    movel([0.494743, -1.360953, -2.580567, -0.770869, 1.570796, 2.065539],accel_mss,speed_ms,0,blend_radius_m)
    movel([0.490867, -1.356572, -2.583531, -0.772287, 1.570796, 2.061664],accel_mss,speed_ms,0,blend_radius_m)
    movel([0.488474, -1.353182, -2.585805, -0.773402, 1.570796, 2.059270],accel_mss,speed_ms,0,blend_radius_m)
    movel([0.485996, -1.348940, -2.588629, -0.774820, 1.570796, 2.056792],accel_mss,speed_ms,0,blend_radius_m)
    movel([0.483593, -1.343799, -2.592018, -0.776572, 1.570796, 2.054390],accel_mss,speed_ms,0,blend_radius_m)
    movel([0.481444, -1.337704, -2.595989, -0.778696, 1.570796, 2.052240],accel_mss,speed_ms,0,blend_radius_m)
    movel([0.480362, -1.333157, -2.598918, -0.780314, 1.570796, 2.051158],accel_mss,speed_ms,0,blend_radius_m)
    movel([0.479844, -1.328776, -2.601714, -0.781898, 1.570796, 2.050640],accel_mss,speed_ms,0,blend_radius_m)
    movel([0.479827, -1.324575, -2.604371, -0.783442, 1.570796, 2.050623],accel_mss,speed_ms,0,blend_radius_m)
    movel([0.480249, -1.320573, -2.606881, -0.784935, 1.570796, 2.051046],accel_mss,speed_ms,0,blend_radius_m)
    movel([0.481050, -1.316778, -2.609241, -0.786370, 1.570796, 2.051846],accel_mss,speed_ms,0,blend_radius_m)
    movel([0.482155, -1.313216, -2.611439, -0.787735, 1.570796, 2.052951],accel_mss,speed_ms,0,blend_radius_m)
    movel([0.483501, -1.309902, -2.613468, -0.789019, 1.570796, 2.054298],accel_mss,speed_ms,0,blend_radius_m)
    movel([0.485016, -1.306856, -2.615321, -0.790212, 1.570796, 2.055813],accel_mss,speed_ms,0,blend_radius_m)
    movel([0.488266, -1.301650, -2.618460, -0.792279, 1.570796, 2.059062],accel_mss,speed_ms,0,blend_radius_m)
    movel([0.491322, -1.297748, -2.620789, -0.793852, 1.570796, 2.062118],accel_mss,speed_ms,0,blend_radius_m)
    movel([0.493591, -1.295306, -2.622237, -0.794846, 1.570796, 2.064387],accel_mss,speed_ms,0,blend_radius_m)
    movel([0.494479, -1.294462, -2.622736, -0.795191, 1.570796, 2.065275],accel_mss,speed_ms,0,blend_radius_m)
    movel([0.498843, -1.290734, -2.624928, -0.796728, 1.570796, 2.069639],accel_mss,speed_ms,0,blend_radius_m)
    movel([0.503178, -1.287586, -2.626765, -0.798039, 1.570796, 2.073975],accel_mss,speed_ms,0,blend_radius_m)
    movel([0.507450, -1.284987, -2.628272, -0.799131, 1.570796, 2.078246],accel_mss,speed_ms,0,blend_radius_m)
    movel([0.511629, -1.282895, -2.629478, -0.800016, 1.570796, 2.082425],accel_mss,speed_ms,0,blend_radius_m)
    movel([0.515682, -1.281272, -2.630411, -0.800706, 1.570796, 2.086478],accel_mss,speed_ms,0,blend_radius_m)
    movel([0.519577, -1.280076, -2.631096, -0.801217, 1.570796, 2.090373],accel_mss,speed_ms,0,blend_radius_m)
    movel([0.523295, -1.279256, -2.631565, -0.801568, 1.570796, 2.094091],accel_mss,speed_ms,0,blend_radius_m)
    movel([0.526799, -1.278773, -2.631841, -0.801776, 1.570796, 2.097596],accel_mss,speed_ms,0,blend_radius_m)
    movel([0.533079, -1.278611, -2.631933, -0.801845, 1.570796, 2.103875],accel_mss,speed_ms,0,blend_radius_m)
    movel([0.538230, -1.279194, -2.631600, -0.801595, 1.570796, 2.109026],accel_mss,speed_ms,0,blend_radius_m)
    movel([0.542077, -1.280114, -2.631074, -0.801201, 1.570796, 2.112873],accel_mss,speed_ms,0,blend_radius_m)
    movel([0.544459, -1.280968, -2.630585, -0.800836, 1.570796, 2.115255],accel_mss,speed_ms,0,blend_radius_m)
    movel([0.550151, -1.282935, -2.629455, -0.799998, 1.570796, 2.120947],accel_mss,speed_ms,0,blend_radius_m)
    movel([0.555976, -1.285582, -2.627927, -0.798880, 1.570796, 2.126773],accel_mss,speed_ms,0,blend_radius_m)
    movel([0.561778, -1.288448, -2.626262, -0.797678, 1.570796, 2.132574],accel_mss,speed_ms,0,blend_radius_m)
    movel([0.567416, -1.291077, -2.624726, -0.796585, 1.570796, 2.138212],accel_mss,speed_ms,0,blend_radius_m)
    movel([0.572766, -1.293010, -2.623591, -0.795787, 1.570796, 2.143562],accel_mss,speed_ms,0,blend_radius_m)
    movel([0.575297, -1.293571, -2.623261, -0.795557, 1.570796, 2.146093],accel_mss,speed_ms,0,blend_radius_m)
    movel([0.577712, -1.293783, -2.623136, -0.795470, 1.570796, 2.148508],accel_mss,speed_ms,0,blend_radius_m)
    movel([0.580003, -1.293588, -2.623251, -0.795550, 1.570796, 2.150799],accel_mss,speed_ms,0,blend_radius_m)
    movel([0.582153, -1.292924, -2.623642, -0.795823, 1.570796, 2.152950],accel_mss,speed_ms,0,blend_radius_m)
    movel([0.584154, -1.291730, -2.624343, -0.796315, 1.570796, 2.154951],accel_mss,speed_ms,0,blend_radius_m)
    movel([0.585992, -1.289947, -2.625388, -0.797054, 1.570796, 2.156788],accel_mss,speed_ms,0,blend_radius_m)
    movel([0.587112, -1.288428, -2.626275, -0.797687, 1.570796, 2.157908],accel_mss,speed_ms,0,blend_radius_m)
    movel([0.587946, -1.286921, -2.627151, -0.798317, 1.570796, 2.158742],accel_mss,speed_ms,0,blend_radius_m)
    movel([0.588873, -1.283945, -2.628874, -0.799571, 1.570796, 2.159669],accel_mss,speed_ms,0,blend_radius_m)
    movel([0.588992, -1.281027, -2.630552, -0.800811, 1.570796, 2.159788],accel_mss,speed_ms,0,blend_radius_m)
    movel([0.588521, -1.278170, -2.632184, -0.802035, 1.570796, 2.159318],accel_mss,speed_ms,0,blend_radius_m)
    movel([0.586712, -1.272683, -2.635291, -0.804415, 1.570796, 2.157508],accel_mss,speed_ms,0,blend_radius_m)
    movel([0.585833, -1.270060, -2.636763, -0.805565, 1.570796, 2.156629],accel_mss,speed_ms,0,blend_radius_m)
    movel([0.585277, -1.267521, -2.638180, -0.806688, 1.570796, 2.156073],accel_mss,speed_ms,0,blend_radius_m)
    movel([0.585264, -1.263324, -2.640505, -0.808560, 1.570796, 2.156061],accel_mss,speed_ms,0,blend_radius_m)
    movel([0.585950, -1.257962, -2.643444, -0.810983, 1.570796, 2.156747],accel_mss,speed_ms,0,blend_radius_m)
    movel([0.587166, -1.252401, -2.646455, -0.813533, 1.570796, 2.157962],accel_mss,speed_ms,0,blend_radius_m)
    movel([0.588725, -1.247651, -2.648998, -0.815741, 1.570796, 2.159522],accel_mss,speed_ms,0,blend_radius_m)
    movel([0.590300, -1.244685, -2.650572, -0.817133, 1.570796, 2.161096],accel_mss,speed_ms,0,blend_radius_m)
    movel([0.592526, -1.241074, -2.652474, -0.818841, 1.570796, 2.163322],accel_mss,speed_ms,0,blend_radius_m)
    movel([0.594616, -1.237629, -2.654274, -0.820486, 1.570796, 2.165412],accel_mss,speed_ms,0,blend_radius_m)
    movel([0.595762, -1.235190, -2.655541, -0.821659, 1.570796, 2.166558],accel_mss,speed_ms,0,blend_radius_m)
    movel([0.595926, -1.232784, -2.656783, -0.822822, 1.570796, 2.166722],accel_mss,speed_ms,0,blend_radius_m)
    movel([0.595622, -1.230098, -2.658162, -0.824129, 1.570796, 2.166418],accel_mss,speed_ms,0,blend_radius_m)
    movel([0.595330, -1.227082, -2.659700, -0.825607, 1.570796, 2.166126],accel_mss,speed_ms,0,blend_radius_m)
    movel([0.595529, -1.223698, -2.661414, -0.827277, 1.570796, 2.166325],accel_mss,speed_ms,0,blend_radius_m)
    movel([0.596137, -1.221575, -2.662482, -0.828331, 1.570796, 2.166934],accel_mss,speed_ms,0,blend_radius_m)
    speed_ms = 0.003
    movel([0.596137, -1.214436, -2.658934, -0.839019, 1.570796, 2.166934],accel_mss,speed_ms,0,blend_radius_m)
    speed_ms = 0.05
    movel([0.596137, -1.187267, -2.644481, -0.880641, 1.570796, 2.166934],accel_mss,speed_ms,0,blend_radius_m)
    #M_RunCode9
    movel([0.481477, -1.280754, -2.594737, -0.836898, 1.570796, 2.052273],accel_mss,speed_ms,0,blend_radius_m)
    #M_RunCode3
    movel([0.481477, -1.306813, -2.607959, -0.797617, 1.570796, 2.052273],accel_mss,speed_ms,0,blend_radius_m)
    speed_ms = 0.003
    movel([0.481477, -1.313612, -2.611195, -0.787582, 1.570796, 2.052273],accel_mss,speed_ms,0,blend_radius_m)
    speed_ms = 0.02
    movel([0.475483, -1.312249, -2.612032, -0.788108, 1.570796, 2.046279],accel_mss,speed_ms,0,blend_radius_m)
    movel([0.469414, -1.311668, -2.612388, -0.788333, 1.570796, 2.040210],accel_mss,speed_ms,0,blend_radius_m)
    movel([0.463339, -1.311775, -2.612323, -0.788291, 1.570796, 2.034136],accel_mss,speed_ms,0,blend_radius_m)
    movel([0.457338, -1.312472, -2.611895, -0.788022, 1.570796, 2.028135],accel_mss,speed_ms,0,blend_radius_m)
    movel([0.451477, -1.313658, -2.611167, -0.787564, 1.570796, 2.022274],accel_mss,speed_ms,0,blend_radius_m)
    movel([0.445825, -1.315241, -2.610191, -0.786957, 1.570796, 2.016621],accel_mss,speed_ms,0,blend_radius_m)
    movel([0.440448, -1.317117, -2.609031, -0.786241, 1.570796, 2.011244],accel_mss,speed_ms,0,blend_radius_m)
    movel([0.435406, -1.319190, -2.607743, -0.785456, 1.570796, 2.006202],accel_mss,speed_ms,0,blend_radius_m)
    movel([0.430761, -1.321359, -2.606390, -0.784640, 1.570796, 2.001558],accel_mss,speed_ms,0,blend_radius_m)
    movel([0.426564, -1.323537, -2.605024, -0.783827, 1.570796, 1.997361],accel_mss,speed_ms,0,blend_radius_m)
    movel([0.419744, -1.327532, -2.602504, -0.782353, 1.570796, 1.990540],accel_mss,speed_ms,0,blend_radius_m)
    movel([0.415357, -1.330446, -2.600651, -0.781291, 1.570796, 1.986153],accel_mss,speed_ms,0,blend_radius_m)
    movel([0.413804, -1.331572, -2.599933, -0.780884, 1.570796, 1.984600],accel_mss,speed_ms,0,blend_radius_m)
    movel([0.411294, -1.333285, -2.598836, -0.780268, 1.570796, 1.982091],accel_mss,speed_ms,0,blend_radius_m)
    movel([0.404926, -1.338198, -2.595668, -0.778522, 1.570796, 1.975722],accel_mss,speed_ms,0,blend_radius_m)
    movel([0.400846, -1.341738, -2.593366, -0.777285, 1.570796, 1.971642],accel_mss,speed_ms,0,blend_radius_m)
    movel([0.396466, -1.345935, -2.590614, -0.775840, 1.570796, 1.967262],accel_mss,speed_ms,0,blend_radius_m)
    movel([0.392003, -1.350733, -2.587438, -0.774218, 1.570796, 1.962799],accel_mss,speed_ms,0,blend_radius_m)
    movel([0.387672, -1.356077, -2.583863, -0.772449, 1.570796, 1.958469],accel_mss,speed_ms,0,blend_radius_m)
    movel([0.383690, -1.361910, -2.579916, -0.770563, 1.570796, 1.954486],accel_mss,speed_ms,0,blend_radius_m)
    movel([0.380257, -1.368174, -2.575624, -0.768591, 1.570796, 1.951053],accel_mss,speed_ms,0,blend_radius_m)
    movel([0.378809, -1.371451, -2.573357, -0.767581, 1.570796, 1.949605],accel_mss,speed_ms,0,blend_radius_m)
    movel([0.377574, -1.374814, -2.571014, -0.766561, 1.570796, 1.948370],accel_mss,speed_ms,0,blend_radius_m)
    movel([0.376569, -1.378261, -2.568596, -0.765532, 1.570796, 1.947365],accel_mss,speed_ms,0,blend_radius_m)
    movel([0.375824, -1.381782, -2.566109, -0.764498, 1.570796, 1.946620],accel_mss,speed_ms,0,blend_radius_m)
    movel([0.375358, -1.385375, -2.563553, -0.763462, 1.570796, 1.946155],accel_mss,speed_ms,0,blend_radius_m)
    movel([0.375192, -1.389030, -2.560933, -0.762426, 1.570796, 1.945988],accel_mss,speed_ms,0,blend_radius_m)
    movel([0.375347, -1.392746, -2.558249, -0.761393, 1.570796, 1.946143],accel_mss,speed_ms,0,blend_radius_m)
    movel([0.375845, -1.396520, -2.555504, -0.760365, 1.570796, 1.946642],accel_mss,speed_ms,0,blend_radius_m)
    movel([0.376703, -1.400348, -2.552698, -0.759343, 1.570796, 1.947499],accel_mss,speed_ms,0,blend_radius_m)
    movel([0.377940, -1.404226, -2.549834, -0.758330, 1.570796, 1.948736],accel_mss,speed_ms,0,blend_radius_m)
    movel([0.379574, -1.408150, -2.546913, -0.757326, 1.570796, 1.950370],accel_mss,speed_ms,0,blend_radius_m)
    movel([0.381625, -1.412125, -2.543930, -0.756333, 1.570796, 1.952421],accel_mss,speed_ms,0,blend_radius_m)
    movel([0.381809, -1.412419, -2.543709, -0.756261, 1.570796, 1.952606],accel_mss,speed_ms,0,blend_radius_m)
    movel([0.384472, -1.415938, -2.541048, -0.755403, 1.570796, 1.955269],accel_mss,speed_ms,0,blend_radius_m)
    movel([0.387226, -1.419017, -2.538705, -0.754667, 1.570796, 1.958022],accel_mss,speed_ms,0,blend_radius_m)
    movel([0.390061, -1.421682, -2.536665, -0.754042, 1.570796, 1.960857],accel_mss,speed_ms,0,blend_radius_m)
    movel([0.392964, -1.423958, -2.534915, -0.753516, 1.570796, 1.963760],accel_mss,speed_ms,0,blend_radius_m)
    movel([0.395929, -1.425869, -2.533439, -0.753081, 1.570796, 1.966725],accel_mss,speed_ms,0,blend_radius_m)
    movel([0.398943, -1.427440, -2.532222, -0.752727, 1.570796, 1.969740],accel_mss,speed_ms,0,blend_radius_m)
    movel([0.401999, -1.428693, -2.531249, -0.752447, 1.570796, 1.972795],accel_mss,speed_ms,0,blend_radius_m)
    movel([0.405084, -1.429647, -2.530506, -0.752236, 1.570796, 1.975880],accel_mss,speed_ms,0,blend_radius_m)
    movel([0.408191, -1.430327, -2.529976, -0.752086, 1.570796, 1.978987],accel_mss,speed_ms,0,blend_radius_m)
    movel([0.411305, -1.430753, -2.529643, -0.751993, 1.570796, 1.982101],accel_mss,speed_ms,0,blend_radius_m)
    movel([0.414421, -1.430943, -2.529495, -0.751951, 1.570796, 1.985217],accel_mss,speed_ms,0,blend_radius_m)
    movel([0.417523, -1.430920, -2.529513, -0.751956, 1.570796, 1.988320],accel_mss,speed_ms,0,blend_radius_m)
    movel([0.423649, -1.430314, -2.529986, -0.752089, 1.570796, 1.994445],accel_mss,speed_ms,0,blend_radius_m)
    movel([0.429591, -1.429088, -2.530942, -0.752360, 1.570796, 2.000387],accel_mss,speed_ms,0,blend_radius_m)
    movel([0.435253, -1.427402, -2.532251, -0.752735, 1.570796, 2.006049],accel_mss,speed_ms,0,blend_radius_m)
    movel([0.440532, -1.425412, -2.533793, -0.753184, 1.570796, 2.011328],accel_mss,speed_ms,0,blend_radius_m)
    movel([0.445320, -1.423278, -2.535439, -0.753672, 1.570796, 2.016117],accel_mss,speed_ms,0,blend_radius_m)
    movel([0.449508, -1.421159, -2.537067, -0.754164, 1.570796, 2.020304],accel_mss,speed_ms,0,blend_radius_m)
    movel([0.455599, -1.417624, -2.539766, -0.754998, 1.570796, 2.026395],accel_mss,speed_ms,0,blend_radius_m)
    movel([0.457844, -1.416144, -2.540891, -0.755353, 1.570796, 2.028641],accel_mss,speed_ms,0,blend_radius_m)
    movel([0.459221, -1.415285, -2.541543, -0.755561, 1.570796, 2.030018],accel_mss,speed_ms,0,blend_radius_m)
    movel([0.462946, -1.412761, -2.543451, -0.756177, 1.570796, 2.033742],accel_mss,speed_ms,0,blend_radius_m)
    movel([0.468426, -1.408636, -2.546549, -0.757204, 1.570796, 2.039222],accel_mss,speed_ms,0,blend_radius_m)
    movel([0.475077, -1.402961, -2.550771, -0.758658, 1.570796, 2.045874],accel_mss,speed_ms,0,blend_radius_m)
    movel([0.478659, -1.399552, -2.553283, -0.759554, 1.570796, 2.049456],accel_mss,speed_ms,0,blend_radius_m)
    movel([0.482313, -1.395770, -2.556051, -0.760568, 1.570796, 2.053109],accel_mss,speed_ms,0,blend_radius_m)
    movel([0.485966, -1.391611, -2.559071, -0.761707, 1.570796, 2.056763],accel_mss,speed_ms,0,blend_radius_m)
    movel([0.489543, -1.387078, -2.562334, -0.762977, 1.570796, 2.060340],accel_mss,speed_ms,0,blend_radius_m)
    movel([0.492966, -1.382172, -2.565833, -0.764385, 1.570796, 2.063763],accel_mss,speed_ms,0,blend_radius_m)
    movel([0.496159, -1.376887, -2.569562, -0.765940, 1.570796, 2.066955],accel_mss,speed_ms,0,blend_radius_m)
    movel([0.499041, -1.371225, -2.573514, -0.767650, 1.570796, 2.069837],accel_mss,speed_ms,0,blend_radius_m)
    movel([0.501524, -1.365181, -2.577682, -0.769526, 1.570796, 2.072320],accel_mss,speed_ms,0,blend_radius_m)
    speed_ms = 0.003
    movel([0.501524, -1.358625, -2.574619, -0.779145, 1.570796, 2.072320],accel_mss,speed_ms,0,blend_radius_m)
    speed_ms = 0.05
    movel([0.501524, -1.333410, -2.562080, -0.816900, 1.570796, 2.072320],accel_mss,speed_ms,0,blend_radius_m)
    #M_RunCode9
    movel([0.476373, -1.327819, -2.565716, -0.818854, 1.570796, 2.047169],accel_mss,speed_ms,0,blend_radius_m)
    #M_RunCode3
    # logo 1
    movel([0.476373, -1.353130, -2.578327, -0.780932, 1.570796, 2.047169],accel_mss,speed_ms,0,blend_radius_m)
    speed_ms = 0.003
    movel([0.476373, -1.359713, -2.581408, -0.771267, 1.570796, 2.047169],accel_mss,speed_ms,0,blend_radius_m)
    speed_ms = 0.007
    movel([0.474310, -1.362233, -2.579696, -0.770460, 1.570796, 2.045106],accel_mss,speed_ms,0,blend_radius_m)
    movel([0.471928, -1.364476, -2.578165, -0.769748, 1.570796, 2.042725],accel_mss,speed_ms,0,blend_radius_m)
    movel([0.469307, -1.366396, -2.576848, -0.769145, 1.570796, 2.040104],accel_mss,speed_ms,0,blend_radius_m)
    movel([0.466525, -1.367946, -2.575781, -0.768662, 1.570796, 2.037321],accel_mss,speed_ms,0,blend_radius_m)
    movel([0.463658, -1.369079, -2.574999, -0.768310, 1.570796, 2.034454],accel_mss,speed_ms,0,blend_radius_m)
    movel([0.460782, -1.369748, -2.574537, -0.768104, 1.570796, 2.031579],accel_mss,speed_ms,0,blend_radius_m)
    movel([0.457972, -1.369904, -2.574429, -0.768056, 1.570796, 2.028768],accel_mss,speed_ms,0,blend_radius_m)
    movel([0.457932, -1.369900, -2.574432, -0.768057, 1.570796, 2.028729],accel_mss,speed_ms,0,blend_radius_m)
    movel([0.451919, -1.369659, -2.574599, -0.768131, 1.570796, 2.022716],accel_mss,speed_ms,0,blend_radius_m)
    movel([0.447534, -1.378826, -2.568198, -0.765365, 1.570796, 2.018330],accel_mss,speed_ms,0,blend_radius_m)
    movel([0.440352, -1.378589, -2.568365, -0.765435, 1.570796, 2.011148],accel_mss,speed_ms,0,blend_radius_m)
    movel([0.452694, -1.352529, -2.586241, -0.773619, 1.570796, 2.023490],accel_mss,speed_ms,0,blend_radius_m)
    movel([0.460066, -1.352777, -2.586076, -0.773536, 1.570796, 2.030863],accel_mss,speed_ms,0,blend_radius_m)
    movel([0.455511, -1.362196, -2.579722, -0.770472, 1.570796, 2.026308],accel_mss,speed_ms,0,blend_radius_m)
    movel([0.461641, -1.362440, -2.579555, -0.770394, 1.570796, 2.032437],accel_mss,speed_ms,0,blend_radius_m)
    movel([0.462915, -1.362365, -2.579606, -0.770418, 1.570796, 2.033711],accel_mss,speed_ms,0,blend_radius_m)
    movel([0.464229, -1.362050, -2.579821, -0.770518, 1.570796, 2.035025],accel_mss,speed_ms,0,blend_radius_m)
    movel([0.465545, -1.361519, -2.580182, -0.770688, 1.570796, 2.036342],accel_mss,speed_ms,0,blend_radius_m)
    movel([0.466825, -1.360800, -2.580671, -0.770918, 1.570796, 2.037621],accel_mss,speed_ms,0,blend_radius_m)
    movel([0.468029, -1.359912, -2.581273, -0.771203, 1.570796, 2.038826],accel_mss,speed_ms,0,blend_radius_m)
    movel([0.469120, -1.358883, -2.581970, -0.771535, 1.570796, 2.039916],accel_mss,speed_ms,0,blend_radius_m)
    movel([0.470058, -1.357734, -2.582747, -0.771908, 1.570796, 2.040854],accel_mss,speed_ms,0,blend_radius_m)
    movel([0.470803, -1.356496, -2.583581, -0.772312, 1.570796, 2.041600],accel_mss,speed_ms,0,blend_radius_m)
    movel([0.471301, -1.355238, -2.584427, -0.772724, 1.570796, 2.042097],accel_mss,speed_ms,0,blend_radius_m)
    movel([0.471534, -1.354042, -2.585229, -0.773118, 1.570796, 2.042330],accel_mss,speed_ms,0,blend_radius_m)
    movel([0.471237, -1.351960, -2.586621, -0.773808, 1.570796, 2.042033],accel_mss,speed_ms,0,blend_radius_m)
    movel([0.470729, -1.351133, -2.587172, -0.774084, 1.570796, 2.041526],accel_mss,speed_ms,0,blend_radius_m)
    movel([0.469993, -1.350487, -2.587602, -0.774300, 1.570796, 2.040790],accel_mss,speed_ms,0,blend_radius_m)
    movel([0.469039, -1.350056, -2.587888, -0.774445, 1.570796, 2.039835],accel_mss,speed_ms,0,blend_radius_m)
    movel([0.467881, -1.349870, -2.588012, -0.774507, 1.570796, 2.038677],accel_mss,speed_ms,0,blend_radius_m)
    movel([0.443597, -1.349099, -2.588523, -0.774767, 1.570796, 2.014394],accel_mss,speed_ms,0,blend_radius_m)
    movel([0.443513, -1.346849, -2.590012, -0.775529, 1.570796, 2.014310],accel_mss,speed_ms,0,blend_radius_m)
    movel([0.443026, -1.344797, -2.591362, -0.776229, 1.570796, 2.013822],accel_mss,speed_ms,0,blend_radius_m)
    movel([0.442144, -1.342981, -2.592554, -0.776855, 1.570796, 2.012940],accel_mss,speed_ms,0,blend_radius_m)
    movel([0.440882, -1.341431, -2.593566, -0.777391, 1.570796, 2.011678],accel_mss,speed_ms,0,blend_radius_m)
    movel([0.471495, -1.342312, -2.592991, -0.777086, 1.570796, 2.042292],accel_mss,speed_ms,0,blend_radius_m)
    movel([0.474100, -1.342726, -2.592720, -0.776942, 1.570796, 2.044896],accel_mss,speed_ms,0,blend_radius_m)
    movel([0.476247, -1.343673, -2.592101, -0.776616, 1.570796, 2.047043],accel_mss,speed_ms,0,blend_radius_m)
    movel([0.477903, -1.345091, -2.591169, -0.776129, 1.570796, 2.048699],accel_mss,speed_ms,0,blend_radius_m)
    movel([0.479042, -1.346916, -2.589967, -0.775506, 1.570796, 2.049839],accel_mss,speed_ms,0,blend_radius_m)
    movel([0.479649, -1.349080, -2.588536, -0.774773, 1.570796, 2.050446],accel_mss,speed_ms,0,blend_radius_m)
    movel([0.479696, -1.351517, -2.586917, -0.773956, 1.570796, 2.050493],accel_mss,speed_ms,0,blend_radius_m)
    movel([0.479166, -1.354167, -2.585146, -0.773076, 1.570796, 2.049963],accel_mss,speed_ms,0,blend_radius_m)
    movel([0.478036, -1.356962, -2.583268, -0.772159, 1.570796, 2.048833],accel_mss,speed_ms,0,blend_radius_m)
    movel([0.476373, -1.359713, -2.581408, -0.771267, 1.570796, 2.047169],accel_mss,speed_ms,0,blend_radius_m)
    speed_ms = 0.003
    movel([0.476373, -1.353130, -2.578327, -0.780932, 1.570796, 2.047169],accel_mss,speed_ms,0,blend_radius_m)
    speed_ms = 0.05
    movel([0.476373, -1.327819, -2.565716, -0.818854, 1.570796, 2.047169],accel_mss,speed_ms,0,blend_radius_m)
    #M_RunCode9
    movel([0.473102, -1.335045, -2.561009, -0.816336, 1.570796, 2.043899],accel_mss,speed_ms,0,blend_radius_m)
    #M_RunCode3
    movel([0.473102, -1.360231, -2.573527, -0.778631, 1.570796, 2.043899],accel_mss,speed_ms,0,blend_radius_m)
    speed_ms = 0.003
    movel([0.473102, -1.366779, -2.576585, -0.769025, 1.570796, 2.043899],accel_mss,speed_ms,0,blend_radius_m)
    speed_ms = 0.007
    movel([0.458507, -1.396201, -2.555737, -0.760451, 1.570796, 2.029303],accel_mss,speed_ms,0,blend_radius_m)
    movel([0.456968, -1.398783, -2.553848, -0.759758, 1.570796, 2.027764],accel_mss,speed_ms,0,blend_radius_m)
    movel([0.455035, -1.401150, -2.552107, -0.759132, 1.570796, 2.025832],accel_mss,speed_ms,0,blend_radius_m)
    movel([0.452787, -1.403260, -2.550549, -0.758580, 1.570796, 2.023584],accel_mss,speed_ms,0,blend_radius_m)
    movel([0.450300, -1.405068, -2.549208, -0.758112, 1.570796, 2.021097],accel_mss,speed_ms,0,blend_radius_m)
    movel([0.447651, -1.406528, -2.548123, -0.757738, 1.570796, 2.018447],accel_mss,speed_ms,0,blend_radius_m)
    movel([0.444911, -1.407596, -2.547326, -0.757467, 1.570796, 2.015707],accel_mss,speed_ms,0,blend_radius_m)
    movel([0.442156, -1.408228, -2.546854, -0.757307, 1.570796, 2.012953],accel_mss,speed_ms,0,blend_radius_m)
    movel([0.439456, -1.408377, -2.546743, -0.757269, 1.570796, 2.010252],accel_mss,speed_ms,0,blend_radius_m)
    movel([0.436993, -1.408020, -2.547010, -0.757359, 1.570796, 2.007790],accel_mss,speed_ms,0,blend_radius_m)
    movel([0.434931, -1.407193, -2.547627, -0.757569, 1.570796, 2.005727],accel_mss,speed_ms,0,blend_radius_m)
    movel([0.433292, -1.405948, -2.548555, -0.757887, 1.570796, 2.004089],accel_mss,speed_ms,0,blend_radius_m)
    movel([0.432112, -1.404329, -2.549757, -0.758303, 1.570796, 2.002908],accel_mss,speed_ms,0,blend_radius_m)
    movel([0.431417, -1.402389, -2.551193, -0.758807, 1.570796, 2.002213],accel_mss,speed_ms,0,blend_radius_m)
    movel([0.431235, -1.400175, -2.552825, -0.759389, 1.570796, 2.002031],accel_mss,speed_ms,0,blend_radius_m)
    movel([0.431603, -1.397735, -2.554616, -0.760038, 1.570796, 2.002399],accel_mss,speed_ms,0,blend_radius_m)
    movel([0.432553, -1.395118, -2.556526, -0.760745, 1.570796, 2.003349],accel_mss,speed_ms,0,blend_radius_m)
    movel([0.432568, -1.395085, -2.556551, -0.760754, 1.570796, 2.003365],accel_mss,speed_ms,0,blend_radius_m)
    movel([0.435306, -1.389209, -2.560804, -0.762376, 1.570796, 2.006103],accel_mss,speed_ms,0,blend_radius_m)
    movel([0.426293, -1.388998, -2.560956, -0.762435, 1.570796, 1.997090],accel_mss,speed_ms,0,blend_radius_m)
    movel([0.429574, -1.381850, -2.566061, -0.764478, 1.570796, 2.000371],accel_mss,speed_ms,0,blend_radius_m)
    movel([0.454905, -1.382667, -2.565481, -0.764241, 1.570796, 2.025702],accel_mss,speed_ms,0,blend_radius_m)
    movel([0.451457, -1.389789, -2.560386, -0.762214, 1.570796, 2.022253],accel_mss,speed_ms,0,blend_radius_m)
    movel([0.442518, -1.389431, -2.560644, -0.762314, 1.570796, 2.013314],accel_mss,speed_ms,0,blend_radius_m)
    movel([0.439706, -1.395372, -2.556341, -0.760676, 1.570796, 2.010502],accel_mss,speed_ms,0,blend_radius_m)
    movel([0.439274, -1.396549, -2.555483, -0.760357, 1.570796, 2.010070],accel_mss,speed_ms,0,blend_radius_m)
    movel([0.439102, -1.397659, -2.554672, -0.760059, 1.570796, 2.009898],accel_mss,speed_ms,0,blend_radius_m)
    movel([0.439181, -1.398675, -2.553927, -0.759787, 1.570796, 2.009977],accel_mss,speed_ms,0,blend_radius_m)
    movel([0.439493, -1.399573, -2.553268, -0.759548, 1.570796, 2.010289],accel_mss,speed_ms,0,blend_radius_m)
    movel([0.440027, -1.400324, -2.552715, -0.759349, 1.570796, 2.010823],accel_mss,speed_ms,0,blend_radius_m)
    movel([0.440767, -1.400907, -2.552286, -0.759195, 1.570796, 2.011563],accel_mss,speed_ms,0,blend_radius_m)
    movel([0.441701, -1.401292, -2.552003, -0.759094, 1.570796, 2.012498],accel_mss,speed_ms,0,blend_radius_m)
    movel([0.442814, -1.401458, -2.551881, -0.759051, 1.570796, 2.013610],accel_mss,speed_ms,0,blend_radius_m)
    movel([0.444039, -1.401392, -2.551929, -0.759068, 1.570796, 2.014835],accel_mss,speed_ms,0,blend_radius_m)
    movel([0.445293, -1.401105, -2.552140, -0.759143, 1.570796, 2.016090],accel_mss,speed_ms,0,blend_radius_m)
    movel([0.447761, -1.399954, -2.552988, -0.759447, 1.570796, 2.018558],accel_mss,speed_ms,0,blend_radius_m)
    movel([0.448900, -1.399134, -2.553590, -0.759665, 1.570796, 2.019696],accel_mss,speed_ms,0,blend_radius_m)
    movel([0.449926, -1.398177, -2.554292, -0.759920, 1.570796, 2.020722],accel_mss,speed_ms,0,blend_radius_m)
    movel([0.450799, -1.397108, -2.555074, -0.760206, 1.570796, 2.021596],accel_mss,speed_ms,0,blend_radius_m)
    movel([0.451489, -1.395945, -2.555923, -0.760520, 1.570796, 2.022286],accel_mss,speed_ms,0,blend_radius_m)
    movel([0.462953, -1.372486, -2.572638, -0.767266, 1.570796, 2.033749],accel_mss,speed_ms,0,blend_radius_m)
    movel([0.465601, -1.371494, -2.573327, -0.767568, 1.570796, 2.036397],accel_mss,speed_ms,0,blend_radius_m)
    movel([0.468204, -1.370195, -2.574227, -0.767966, 1.570796, 2.039000],accel_mss,speed_ms,0,blend_radius_m)
    movel([0.470719, -1.368615, -2.575320, -0.768454, 1.570796, 2.041515],accel_mss,speed_ms,0,blend_radius_m)
    movel([0.473102, -1.366779, -2.576585, -0.769025, 1.570796, 2.043899],accel_mss,speed_ms,0,blend_radius_m)
    speed_ms = 0.003
    movel([0.473102, -1.360231, -2.573527, -0.778631, 1.570796, 2.043899],accel_mss,speed_ms,0,blend_radius_m)
    speed_ms = 0.05
    movel([0.473102, -1.335045, -2.561009, -0.816336, 1.570796, 2.043899],accel_mss,speed_ms,0,blend_radius_m)
    #M_RunCode9
    movel([0.430338, -1.340996, -2.557079, -0.814314, 1.570796, 2.001135],accel_mss,speed_ms,0,blend_radius_m)
    #M_RunCode3
    movel([0.430338, -1.366079, -2.569521, -0.776789, 1.570796, 2.001135],accel_mss,speed_ms,0,blend_radius_m)
    speed_ms = 0.003
    movel([0.430338, -1.372597, -2.572560, -0.767232, 1.570796, 2.001135],accel_mss,speed_ms,0,blend_radius_m)
    speed_ms = 0.007
    movel([0.418840, -1.397865, -2.554520, -0.760003, 1.570796, 1.989636],accel_mss,speed_ms,0,blend_radius_m)
    movel([0.411716, -1.397782, -2.554581, -0.760026, 1.570796, 1.982512],accel_mss,speed_ms,0,blend_radius_m)
    movel([0.415691, -1.388881, -2.561040, -0.762468, 1.570796, 1.986487],accel_mss,speed_ms,0,blend_radius_m)
    movel([0.409628, -1.388847, -2.561065, -0.762478, 1.570796, 1.980424],accel_mss,speed_ms,0,blend_radius_m)
    movel([0.408368, -1.388966, -2.560979, -0.762444, 1.570796, 1.979164],accel_mss,speed_ms,0,blend_radius_m)
    movel([0.407083, -1.389316, -2.560727, -0.762346, 1.570796, 1.977880],accel_mss,speed_ms,0,blend_radius_m)
    movel([0.405815, -1.389871, -2.560327, -0.762191, 1.570796, 1.976612],accel_mss,speed_ms,0,blend_radius_m)
    movel([0.404599, -1.390603, -2.559799, -0.761987, 1.570796, 1.975395],accel_mss,speed_ms,0,blend_radius_m)
    movel([0.403472, -1.391486, -2.559161, -0.761741, 1.570796, 1.974268],accel_mss,speed_ms,0,blend_radius_m)
    movel([0.402472, -1.392493, -2.558433, -0.761463, 1.570796, 1.973269],accel_mss,speed_ms,0,blend_radius_m)
    movel([0.401637, -1.393599, -2.557631, -0.761159, 1.570796, 1.972433],accel_mss,speed_ms,0,blend_radius_m)
    movel([0.401005, -1.394776, -2.556775, -0.760838, 1.570796, 1.971801],accel_mss,speed_ms,0,blend_radius_m)
    movel([0.400616, -1.395953, -2.555918, -0.760518, 1.570796, 1.971412],accel_mss,speed_ms,0,blend_radius_m)
    movel([0.400482, -1.397053, -2.555114, -0.760221, 1.570796, 1.971279],accel_mss,speed_ms,0,blend_radius_m)
    movel([0.400938, -1.398930, -2.553740, -0.759719, 1.570796, 1.971735],accel_mss,speed_ms,0,blend_radius_m)
    movel([0.401499, -1.399656, -2.553207, -0.759526, 1.570796, 1.972295],accel_mss,speed_ms,0,blend_radius_m)
    movel([0.402263, -1.400207, -2.552801, -0.759380, 1.570796, 1.973059],accel_mss,speed_ms,0,blend_radius_m)
    movel([0.403215, -1.400560, -2.552542, -0.759287, 1.570796, 1.974012],accel_mss,speed_ms,0,blend_radius_m)
    movel([0.404350, -1.400685, -2.552450, -0.759254, 1.570796, 1.975146],accel_mss,speed_ms,0,blend_radius_m)
    movel([0.427605, -1.400998, -2.552219, -0.759172, 1.570796, 1.998401],accel_mss,speed_ms,0,blend_radius_m)
    movel([0.427724, -1.403075, -2.550686, -0.758628, 1.570796, 1.998520],accel_mss,speed_ms,0,blend_radius_m)
    movel([0.428219, -1.404958, -2.549290, -0.758141, 1.570796, 1.999015],accel_mss,speed_ms,0,blend_radius_m)
    movel([0.429069, -1.406625, -2.548051, -0.757714, 1.570796, 1.999865],accel_mss,speed_ms,0,blend_radius_m)
    movel([0.430259, -1.408049, -2.546988, -0.757352, 1.570796, 2.001055],accel_mss,speed_ms,0,blend_radius_m)
    movel([0.401447, -1.407575, -2.547342, -0.757472, 1.570796, 1.972243],accel_mss,speed_ms,0,blend_radius_m)
    movel([0.398929, -1.407313, -2.547537, -0.757538, 1.570796, 1.969725],accel_mss,speed_ms,0,blend_radius_m)
    movel([0.396797, -1.406575, -2.548088, -0.757726, 1.570796, 1.967594],accel_mss,speed_ms,0,blend_radius_m)
    movel([0.395080, -1.405404, -2.548959, -0.758026, 1.570796, 1.965877],accel_mss,speed_ms,0,blend_radius_m)
    movel([0.393810, -1.403852, -2.550111, -0.758426, 1.570796, 1.964607],accel_mss,speed_ms,0,blend_radius_m)
    movel([0.393017, -1.401963, -2.551508, -0.758918, 1.570796, 1.963813],accel_mss,speed_ms,0,blend_radius_m)
    movel([0.392732, -1.399786, -2.553111, -0.759492, 1.570796, 1.963528],accel_mss,speed_ms,0,blend_radius_m)
    movel([0.392993, -1.397371, -2.554882, -0.760136, 1.570796, 1.963790],accel_mss,speed_ms,0,blend_radius_m)
    movel([0.393836, -1.394764, -2.556784, -0.760841, 1.570796, 1.964632],accel_mss,speed_ms,0,blend_radius_m)
    movel([0.395222, -1.392143, -2.558687, -0.761560, 1.570796, 1.966018],accel_mss,speed_ms,0,blend_radius_m)
    movel([0.397044, -1.389685, -2.560462, -0.762243, 1.570796, 1.967840],accel_mss,speed_ms,0,blend_radius_m)
    movel([0.399229, -1.387449, -2.562068, -0.762872, 1.570796, 1.970026],accel_mss,speed_ms,0,blend_radius_m)
    movel([0.401703, -1.385492, -2.563469, -0.763428, 1.570796, 1.972500],accel_mss,speed_ms,0,blend_radius_m)
    movel([0.404383, -1.383869, -2.564626, -0.763894, 1.570796, 1.975179],accel_mss,speed_ms,0,blend_radius_m)
    movel([0.407191, -1.382643, -2.565498, -0.764248, 1.570796, 1.977988],accel_mss,speed_ms,0,blend_radius_m)
    movel([0.410046, -1.381867, -2.566049, -0.764473, 1.570796, 1.980842],accel_mss,speed_ms,0,blend_radius_m)
    movel([0.412863, -1.381600, -2.566238, -0.764551, 1.570796, 1.983659],accel_mss,speed_ms,0,blend_radius_m)
    movel([0.412893, -1.381610, -2.566231, -0.764548, 1.570796, 1.983690],accel_mss,speed_ms,0,blend_radius_m)
    movel([0.418934, -1.381635, -2.566213, -0.764541, 1.570796, 1.989730],accel_mss,speed_ms,0,blend_radius_m)
    movel([0.423040, -1.372509, -2.572622, -0.767259, 1.570796, 1.993836],accel_mss,speed_ms,0,blend_radius_m)
    movel([0.430338, -1.372597, -2.572560, -0.767232, 1.570796, 2.001135],accel_mss,speed_ms,0,blend_radius_m)
    speed_ms = 0.003
    movel([0.430338, -1.366079, -2.569521, -0.776789, 1.570796, 2.001135],accel_mss,speed_ms,0,blend_radius_m)
    speed_ms = 0.05
    movel([0.430338, -1.340996, -2.557079, -0.814314, 1.570796, 2.001135],accel_mss,speed_ms,0,blend_radius_m)
    #M_RunCode9
    movel([0.441221, -1.337598, -2.559328, -0.815462, 1.570796, 2.012017],accel_mss,speed_ms,0,blend_radius_m)
    #M_RunCode3
    movel([0.441221, -1.362741, -2.571814, -0.777835, 1.570796, 2.012017],accel_mss,speed_ms,0,blend_radius_m)
    speed_ms = 0.003
    movel([0.441221, -1.369276, -2.574863, -0.768250, 1.570796, 2.012017],accel_mss,speed_ms,0,blend_radius_m)
    speed_ms = 0.007
    movel([0.415317, -1.368956, -2.575084, -0.768348, 1.570796, 1.986114],accel_mss,speed_ms,0,blend_radius_m)
    movel([0.418598, -1.361578, -2.580142, -0.770669, 1.570796, 1.989395],accel_mss,speed_ms,0,blend_radius_m)
    movel([0.427943, -1.361617, -2.580116, -0.770656, 1.570796, 1.998739],accel_mss,speed_ms,0,blend_radius_m)
    movel([0.430801, -1.355337, -2.584361, -0.772691, 1.570796, 2.001597],accel_mss,speed_ms,0,blend_radius_m)
    movel([0.431246, -1.354083, -2.585202, -0.773104, 1.570796, 2.002042],accel_mss,speed_ms,0,blend_radius_m)
    movel([0.431413, -1.352905, -2.585990, -0.773494, 1.570796, 2.002210],accel_mss,speed_ms,0,blend_radius_m)
    movel([0.431318, -1.351830, -2.586708, -0.773851, 1.570796, 2.002115],accel_mss,speed_ms,0,blend_radius_m)
    movel([0.430976, -1.350885, -2.587337, -0.774167, 1.570796, 2.001773],accel_mss,speed_ms,0,blend_radius_m)
    movel([0.430399, -1.350101, -2.587859, -0.774430, 1.570796, 2.001196],accel_mss,speed_ms,0,blend_radius_m)
    movel([0.429603, -1.349504, -2.588255, -0.774630, 1.570796, 2.000400],accel_mss,speed_ms,0,blend_radius_m)
    movel([0.428599, -1.349124, -2.588507, -0.774758, 1.570796, 1.999395],accel_mss,speed_ms,0,blend_radius_m)
    movel([0.427405, -1.348989, -2.588596, -0.774804, 1.570796, 1.998202],accel_mss,speed_ms,0,blend_radius_m)
    movel([0.426094, -1.349114, -2.588514, -0.774762, 1.570796, 1.996891],accel_mss,speed_ms,0,blend_radius_m)
    movel([0.424752, -1.349478, -2.588272, -0.774639, 1.570796, 1.995548],accel_mss,speed_ms,0,blend_radius_m)
    movel([0.422133, -1.350821, -2.587380, -0.774188, 1.570796, 1.992930],accel_mss,speed_ms,0,blend_radius_m)
    movel([0.420941, -1.351746, -2.586764, -0.773880, 1.570796, 1.991738],accel_mss,speed_ms,0,blend_radius_m)
    movel([0.419877, -1.352806, -2.586056, -0.773527, 1.570796, 1.990673],accel_mss,speed_ms,0,blend_radius_m)
    movel([0.418982, -1.353976, -2.585274, -0.773140, 1.570796, 1.989779],accel_mss,speed_ms,0,blend_radius_m)
    movel([0.418292, -1.355230, -2.584433, -0.772726, 1.570796, 1.989088],accel_mss,speed_ms,0,blend_radius_m)
    movel([0.407677, -1.379350, -2.567829, -0.765210, 1.570796, 1.978473],accel_mss,speed_ms,0,blend_radius_m)
    movel([0.405051, -1.380450, -2.567052, -0.764887, 1.570796, 1.975847],accel_mss,speed_ms,0,blend_radius_m)
    movel([0.402508, -1.381841, -2.566067, -0.764481, 1.570796, 1.973305],accel_mss,speed_ms,0,blend_radius_m)
    movel([0.400092, -1.383495, -2.564892, -0.764002, 1.570796, 1.970888],accel_mss,speed_ms,0,blend_radius_m)
    movel([0.397842, -1.385379, -2.563550, -0.763460, 1.570796, 1.968638],accel_mss,speed_ms,0,blend_radius_m)
    movel([0.410800, -1.355390, -2.584325, -0.772674, 1.570796, 1.981596],accel_mss,speed_ms,0,blend_radius_m)
    movel([0.412299, -1.352599, -2.586195, -0.773596, 1.570796, 1.983095],accel_mss,speed_ms,0,blend_radius_m)
    movel([0.414254, -1.349980, -2.587939, -0.774470, 1.570796, 1.985050],accel_mss,speed_ms,0,blend_radius_m)
    movel([0.416584, -1.347599, -2.589516, -0.775274, 1.570796, 1.987380],accel_mss,speed_ms,0,blend_radius_m)
    movel([0.419203, -1.345515, -2.590891, -0.775983, 1.570796, 1.989999],accel_mss,speed_ms,0,blend_radius_m)
    movel([0.422035, -1.343786, -2.592027, -0.776577, 1.570796, 1.992831],accel_mss,speed_ms,0,blend_radius_m)
    movel([0.424990, -1.342479, -2.592882, -0.777028, 1.570796, 1.995786],accel_mss,speed_ms,0,blend_radius_m)
    movel([0.427980, -1.341654, -2.593421, -0.777314, 1.570796, 1.998777],accel_mss,speed_ms,0,blend_radius_m)
    movel([0.430919, -1.341370, -2.593606, -0.777413, 1.570796, 2.001715],accel_mss,speed_ms,0,blend_radius_m)
    movel([0.433596, -1.341666, -2.593413, -0.777310, 1.570796, 2.004393],accel_mss,speed_ms,0,blend_radius_m)
    movel([0.435830, -1.342507, -2.592864, -0.777018, 1.570796, 2.006626],accel_mss,speed_ms,0,blend_radius_m)
    movel([0.437588, -1.343827, -2.591999, -0.776563, 1.570796, 2.008384],accel_mss,speed_ms,0,blend_radius_m)
    movel([0.438845, -1.345566, -2.590857, -0.775966, 1.570796, 2.009641],accel_mss,speed_ms,0,blend_radius_m)
    movel([0.439571, -1.347661, -2.589475, -0.775253, 1.570796, 2.010367],accel_mss,speed_ms,0,blend_radius_m)
    movel([0.439737, -1.350049, -2.587893, -0.774447, 1.570796, 2.010534],accel_mss,speed_ms,0,blend_radius_m)
    movel([0.439326, -1.352672, -2.586146, -0.773571, 1.570796, 2.010123],accel_mss,speed_ms,0,blend_radius_m)
    movel([0.438308, -1.355467, -2.584274, -0.772649, 1.570796, 2.009105],accel_mss,speed_ms,0,blend_radius_m)
    movel([0.438291, -1.355505, -2.584248, -0.772636, 1.570796, 2.009087],accel_mss,speed_ms,0,blend_radius_m)
    movel([0.435424, -1.361712, -2.580051, -0.770626, 1.570796, 2.006220],accel_mss,speed_ms,0,blend_radius_m)
    movel([0.444685, -1.361908, -2.579917, -0.770563, 1.570796, 2.015481],accel_mss,speed_ms,0,blend_radius_m)
    movel([0.441221, -1.369276, -2.574863, -0.768250, 1.570796, 2.012017],accel_mss,speed_ms,0,blend_radius_m)
    speed_ms = 0.003
    movel([0.441221, -1.362741, -2.571814, -0.777835, 1.570796, 2.012017],accel_mss,speed_ms,0,blend_radius_m)
    speed_ms = 0.05
    movel([0.441221, -1.337598, -2.559328, -0.815462, 1.570796, 2.012017],accel_mss,speed_ms,0,blend_radius_m)
    #M_RunCode9
    movel([0.389142, -1.390622, -2.522452, -0.799315, 1.570796, 1.959938],accel_mss,speed_ms,0,blend_radius_m)
    #M_RunCode3
    movel([0.389142, -1.414788, -2.534268, -0.763332, 1.570796, 1.959938],accel_mss,speed_ms,0,blend_radius_m)
    speed_ms = 0.003
    movel([0.389142, -1.421050, -2.537150, -0.754189, 1.570796, 1.959938],accel_mss,speed_ms,0,blend_radius_m)
    speed_ms = 0.02
    movel([0.391932, -1.423805, -2.535032, -0.753551, 1.570796, 1.962728],accel_mss,speed_ms,0,blend_radius_m)
    movel([0.396326, -1.427031, -2.532539, -0.752819, 1.570796, 1.967122],accel_mss,speed_ms,0,blend_radius_m)
    movel([0.401833, -1.430438, -2.529890, -0.752062, 1.570796, 1.972629],accel_mss,speed_ms,0,blend_radius_m)
    movel([0.407982, -1.433735, -2.527308, -0.751346, 1.570796, 1.978778],accel_mss,speed_ms,0,blend_radius_m)
    movel([0.414319, -1.436617, -2.525038, -0.750734, 1.570796, 1.985115],accel_mss,speed_ms,0,blend_radius_m)
    movel([0.420411, -1.438773, -2.523332, -0.750284, 1.570796, 1.991207],accel_mss,speed_ms,0,blend_radius_m)
    movel([0.423236, -1.439476, -2.522774, -0.750139, 1.570796, 1.994032],accel_mss,speed_ms,0,blend_radius_m)
    movel([0.425844, -1.439877, -2.522456, -0.750056, 1.570796, 1.996640],accel_mss,speed_ms,0,blend_radius_m)
    movel([0.428187, -1.439928, -2.522416, -0.750046, 1.570796, 1.998984],accel_mss,speed_ms,0,blend_radius_m)
    movel([0.430213, -1.439588, -2.522685, -0.750116, 1.570796, 2.001009],accel_mss,speed_ms,0,blend_radius_m)
    movel([0.431775, -1.438861, -2.523262, -0.750266, 1.570796, 2.002571],accel_mss,speed_ms,0,blend_radius_m)
    movel([0.432204, -1.438420, -2.523612, -0.750357, 1.570796, 2.003000],accel_mss,speed_ms,0,blend_radius_m)
    movel([0.432421, -1.437932, -2.523999, -0.750459, 1.570796, 2.003217],accel_mss,speed_ms,0,blend_radius_m)
    movel([0.432300, -1.436833, -2.524868, -0.750688, 1.570796, 2.003096],accel_mss,speed_ms,0,blend_radius_m)
    movel([0.431561, -1.435604, -2.525838, -0.750947, 1.570796, 2.002357],accel_mss,speed_ms,0,blend_radius_m)
    movel([0.428808, -1.432903, -2.527961, -0.751525, 1.570796, 1.999604],accel_mss,speed_ms,0,blend_radius_m)
    movel([0.425359, -1.430121, -2.530136, -0.752131, 1.570796, 1.996155],accel_mss,speed_ms,0,blend_radius_m)
    speed_ms = 0.003
    movel([0.425359, -1.423910, -2.527283, -0.761196, 1.570796, 1.996155],accel_mss,speed_ms,0,blend_radius_m)
    speed_ms = 0.05
    movel([0.425359, -1.399925, -2.515581, -0.796882, 1.570796, 1.996155],accel_mss,speed_ms,0,blend_radius_m)
    #M_RunCode9
    movel([0.559070, -1.327377, -2.566002, -0.819010, 1.570796, 2.129866],accel_mss,speed_ms,0,blend_radius_m)
    #M_RunCode3
    movel([0.559070, -1.352695, -2.578619, -0.781075, 1.570796, 2.129866],accel_mss,speed_ms,0,blend_radius_m)
    speed_ms = 0.003
    movel([0.559070, -1.359280, -2.581702, -0.771407, 1.570796, 2.129866],accel_mss,speed_ms,0,blend_radius_m)
    speed_ms = 0.02
    movel([0.559167, -1.358339, -2.582339, -0.771712, 1.570796, 2.129963],accel_mss,speed_ms,0,blend_radius_m)
    movel([0.559899, -1.357412, -2.582964, -0.772013, 1.570796, 2.130696],accel_mss,speed_ms,0,blend_radius_m)
    movel([0.560267, -1.357112, -2.583167, -0.772111, 1.570796, 2.131064],accel_mss,speed_ms,0,blend_radius_m)
    movel([0.563069, -1.354807, -2.584716, -0.772865, 1.570796, 2.133866],accel_mss,speed_ms,0,blend_radius_m)
    movel([0.565842, -1.352342, -2.586366, -0.773681, 1.570796, 2.136638],accel_mss,speed_ms,0,blend_radius_m)
    movel([0.568362, -1.349708, -2.588120, -0.774562, 1.570796, 2.139158],accel_mss,speed_ms,0,blend_radius_m)
    movel([0.570408, -1.346896, -2.589980, -0.775512, 1.570796, 2.141204],accel_mss,speed_ms,0,blend_radius_m)
    movel([0.571781, -1.343969, -2.591906, -0.776514, 1.570796, 2.142577],accel_mss,speed_ms,0,blend_radius_m)
    movel([0.572570, -1.341024, -2.593832, -0.777533, 1.570796, 2.143367],accel_mss,speed_ms,0,blend_radius_m)
    movel([0.572969, -1.338121, -2.595718, -0.778549, 1.570796, 2.143765],accel_mss,speed_ms,0,blend_radius_m)
    movel([0.573163, -1.335329, -2.597522, -0.779538, 1.570796, 2.143960],accel_mss,speed_ms,0,blend_radius_m)
    movel([0.573184, -1.334942, -2.597772, -0.779675, 1.570796, 2.143981],accel_mss,speed_ms,0,blend_radius_m)
    movel([0.573598, -1.333925, -2.598425, -0.780038, 1.570796, 2.144394],accel_mss,speed_ms,0,blend_radius_m)
    movel([0.574570, -1.333076, -2.598970, -0.780343, 1.570796, 2.145367],accel_mss,speed_ms,0,blend_radius_m)
    movel([0.575690, -1.332743, -2.599184, -0.780462, 1.570796, 2.146486],accel_mss,speed_ms,0,blend_radius_m)
    movel([0.576481, -1.333080, -2.598968, -0.780341, 1.570796, 2.147277],accel_mss,speed_ms,0,blend_radius_m)
    movel([0.576674, -1.333326, -2.598810, -0.780253, 1.570796, 2.147471],accel_mss,speed_ms,0,blend_radius_m)
    movel([0.578171, -1.335179, -2.597619, -0.779591, 1.570796, 2.148967],accel_mss,speed_ms,0,blend_radius_m)
    movel([0.579867, -1.336921, -2.596495, -0.778973, 1.570796, 2.150663],accel_mss,speed_ms,0,blend_radius_m)
    movel([0.581875, -1.338322, -2.595588, -0.778479, 1.570796, 2.152672],accel_mss,speed_ms,0,blend_radius_m)
    movel([0.584308, -1.339151, -2.595051, -0.778188, 1.570796, 2.155104],accel_mss,speed_ms,0,blend_radius_m)
    movel([0.587184, -1.339241, -2.594992, -0.778156, 1.570796, 2.157980],accel_mss,speed_ms,0,blend_radius_m)
    movel([0.590341, -1.338738, -2.595318, -0.778332, 1.570796, 2.161138],accel_mss,speed_ms,0,blend_radius_m)
    movel([0.593616, -1.337866, -2.595884, -0.778639, 1.570796, 2.164412],accel_mss,speed_ms,0,blend_radius_m)
    movel([0.596851, -1.336843, -2.596546, -0.779000, 1.570796, 2.167648],accel_mss,speed_ms,0,blend_radius_m)
    movel([0.597298, -1.336698, -2.596639, -0.779052, 1.570796, 2.168094],accel_mss,speed_ms,0,blend_radius_m)
    movel([0.598307, -1.336674, -2.596655, -0.779060, 1.570796, 2.169103],accel_mss,speed_ms,0,blend_radius_m)
    movel([0.598843, -1.337291, -2.596256, -0.778842, 1.570796, 2.169640],accel_mss,speed_ms,0,blend_radius_m)
    movel([0.598698, -1.338278, -2.595617, -0.778494, 1.570796, 2.169495],accel_mss,speed_ms,0,blend_radius_m)
    movel([0.597919, -1.339223, -2.595004, -0.778162, 1.570796, 2.168715],accel_mss,speed_ms,0,blend_radius_m)
    movel([0.597540, -1.339521, -2.594810, -0.778058, 1.570796, 2.168337],accel_mss,speed_ms,0,blend_radius_m)
    movel([0.594634, -1.341834, -2.593303, -0.777251, 1.570796, 2.165431],accel_mss,speed_ms,0,blend_radius_m)
    movel([0.591775, -1.344302, -2.591688, -0.776399, 1.570796, 2.162571],accel_mss,speed_ms,0,blend_radius_m)
    movel([0.589189, -1.346930, -2.589958, -0.775501, 1.570796, 2.159986],accel_mss,speed_ms,0,blend_radius_m)
    movel([0.587097, -1.349729, -2.588106, -0.774555, 1.570796, 2.157893],accel_mss,speed_ms,0,blend_radius_m)
    movel([0.585692, -1.352627, -2.586176, -0.773586, 1.570796, 2.156488],accel_mss,speed_ms,0,blend_radius_m)
    movel([0.584871, -1.355526, -2.584234, -0.772629, 1.570796, 2.155667],accel_mss,speed_ms,0,blend_radius_m)
    movel([0.584444, -1.358363, -2.582322, -0.771704, 1.570796, 2.155240],accel_mss,speed_ms,0,blend_radius_m)
    movel([0.584220, -1.361078, -2.580482, -0.770829, 1.570796, 2.155016],accel_mss,speed_ms,0,blend_radius_m)
    movel([0.584188, -1.361482, -2.580207, -0.770699, 1.570796, 2.154984],accel_mss,speed_ms,0,blend_radius_m)
    movel([0.584182, -1.361520, -2.580182, -0.770688, 1.570796, 2.154978],accel_mss,speed_ms,0,blend_radius_m)
    movel([0.584156, -1.361666, -2.580082, -0.770641, 1.570796, 2.154952],accel_mss,speed_ms,0,blend_radius_m)
    movel([0.583701, -1.362541, -2.579486, -0.770362, 1.570796, 2.154498],accel_mss,speed_ms,0,blend_radius_m)
    movel([0.582827, -1.363220, -2.579023, -0.770146, 1.570796, 2.153623],accel_mss,speed_ms,0,blend_radius_m)
    movel([0.581871, -1.363526, -2.578814, -0.770049, 1.570796, 2.152667],accel_mss,speed_ms,0,blend_radius_m)
    movel([0.581132, -1.363306, -2.578964, -0.770118, 1.570796, 2.151929],accel_mss,speed_ms,0,blend_radius_m)
    movel([0.581034, -1.363215, -2.579026, -0.770147, 1.570796, 2.151830],accel_mss,speed_ms,0,blend_radius_m)
    movel([0.581016, -1.363199, -2.579037, -0.770152, 1.570796, 2.151812],accel_mss,speed_ms,0,blend_radius_m)
    movel([0.580985, -1.363161, -2.579064, -0.770165, 1.570796, 2.151781],accel_mss,speed_ms,0,blend_radius_m)
    movel([0.580819, -1.362940, -2.579214, -0.770235, 1.570796, 2.151615],accel_mss,speed_ms,0,blend_radius_m)
    movel([0.579376, -1.361134, -2.580444, -0.770811, 1.570796, 2.150173],accel_mss,speed_ms,0,blend_radius_m)
    movel([0.577727, -1.359433, -2.581598, -0.771358, 1.570796, 2.148524],accel_mss,speed_ms,0,blend_radius_m)
    movel([0.575757, -1.358068, -2.582521, -0.771799, 1.570796, 2.146554],accel_mss,speed_ms,0,blend_radius_m)
    movel([0.573361, -1.357265, -2.583063, -0.772061, 1.570796, 2.144158],accel_mss,speed_ms,0,blend_radius_m)
    movel([0.570534, -1.357192, -2.583113, -0.772085, 1.570796, 2.141330],accel_mss,speed_ms,0,blend_radius_m)
    movel([0.567433, -1.357711, -2.582763, -0.771916, 1.570796, 2.138229],accel_mss,speed_ms,0,blend_radius_m)
    movel([0.564224, -1.358605, -2.582159, -0.771626, 1.570796, 2.135021],accel_mss,speed_ms,0,blend_radius_m)
    movel([0.561069, -1.359652, -2.581450, -0.771287, 1.570796, 2.131865],accel_mss,speed_ms,0,blend_radius_m)
    movel([0.560624, -1.359804, -2.581347, -0.771238, 1.570796, 2.131421],accel_mss,speed_ms,0,blend_radius_m)
    movel([0.559996, -1.359912, -2.581274, -0.771203, 1.570796, 2.130792],accel_mss,speed_ms,0,blend_radius_m)
    movel([0.559486, -1.359792, -2.581355, -0.771242, 1.570796, 2.130283],accel_mss,speed_ms,0,blend_radius_m)
    movel([0.559070, -1.359280, -2.581702, -0.771407, 1.570796, 2.129866],accel_mss,speed_ms,0,blend_radius_m)
    speed_ms = 0.003
    movel([0.559070, -1.352695, -2.578619, -0.781075, 1.570796, 2.129866],accel_mss,speed_ms,0,blend_radius_m)
    speed_ms = 0.05
    movel([0.559070, -1.327377, -2.566002, -0.819010, 1.570796, 2.129866],accel_mss,speed_ms,0,blend_radius_m)
    #M_RunCode9
    movel([0.352418, -1.353819, -2.548453, -0.810117, 1.570796, 1.923214],accel_mss,speed_ms,0,blend_radius_m)
    #M_RunCode3
    movel([0.352418, -1.378674, -2.560731, -0.772984, 1.570796, 1.923214],accel_mss,speed_ms,0,blend_radius_m)
    speed_ms = 0.003
    movel([0.352418, -1.385127, -2.563729, -0.763532, 1.570796, 1.923214],accel_mss,speed_ms,0,blend_radius_m)
    speed_ms = 0.02
    movel([0.352035, -1.385789, -2.563257, -0.763343, 1.570796, 1.922832],accel_mss,speed_ms,0,blend_radius_m)
    movel([0.351818, -1.386016, -2.563094, -0.763279, 1.570796, 1.922615],accel_mss,speed_ms,0,blend_radius_m)
    movel([0.348559, -1.389629, -2.560502, -0.762258, 1.570796, 1.919355],accel_mss,speed_ms,0,blend_radius_m)
    movel([0.347187, -1.391530, -2.559130, -0.761729, 1.570796, 1.917983],accel_mss,speed_ms,0,blend_radius_m)
    movel([0.346205, -1.393460, -2.557732, -0.761197, 1.570796, 1.917001],accel_mss,speed_ms,0,blend_radius_m)
    movel([0.345737, -1.395351, -2.556356, -0.760681, 1.570796, 1.916533],accel_mss,speed_ms,0,blend_radius_m)
    movel([0.345696, -1.397159, -2.555037, -0.760193, 1.570796, 1.916492],accel_mss,speed_ms,0,blend_radius_m)
    movel([0.346285, -1.400500, -2.552586, -0.759303, 1.570796, 1.917081],accel_mss,speed_ms,0,blend_radius_m)
    movel([0.346340, -1.400742, -2.552408, -0.759239, 1.570796, 1.917136],accel_mss,speed_ms,0,blend_radius_m)
    movel([0.346341, -1.400764, -2.552392, -0.759233, 1.570796, 1.917137],accel_mss,speed_ms,0,blend_radius_m)
    movel([0.346350, -1.400854, -2.552326, -0.759210, 1.570796, 1.917146],accel_mss,speed_ms,0,blend_radius_m)
    movel([0.346187, -1.401434, -2.551898, -0.759057, 1.570796, 1.916983],accel_mss,speed_ms,0,blend_radius_m)
    movel([0.345678, -1.401959, -2.551511, -0.758919, 1.570796, 1.916474],accel_mss,speed_ms,0,blend_radius_m)
    movel([0.345038, -1.402279, -2.551275, -0.758836, 1.570796, 1.915835],accel_mss,speed_ms,0,blend_radius_m)
    movel([0.344458, -1.402257, -2.551291, -0.758841, 1.570796, 1.915254],accel_mss,speed_ms,0,blend_radius_m)
    movel([0.344369, -1.402219, -2.551319, -0.758851, 1.570796, 1.915165],accel_mss,speed_ms,0,blend_radius_m)
    movel([0.344351, -1.402211, -2.551325, -0.758853, 1.570796, 1.915148],accel_mss,speed_ms,0,blend_radius_m)
    movel([0.344322, -1.402193, -2.551338, -0.758858, 1.570796, 1.915118],accel_mss,speed_ms,0,blend_radius_m)
    movel([0.344157, -1.402089, -2.551415, -0.758885, 1.570796, 1.914953],accel_mss,speed_ms,0,blend_radius_m)
    movel([0.341237, -1.400482, -2.552600, -0.759308, 1.570796, 1.912033],accel_mss,speed_ms,0,blend_radius_m)
    movel([0.339545, -1.399965, -2.552979, -0.759444, 1.570796, 1.910342],accel_mss,speed_ms,0,blend_radius_m)
    movel([0.337651, -1.399840, -2.553071, -0.759477, 1.570796, 1.908447],accel_mss,speed_ms,0,blend_radius_m)
    movel([0.335582, -1.400202, -2.552806, -0.759382, 1.570796, 1.906378],accel_mss,speed_ms,0,blend_radius_m)
    movel([0.333428, -1.400947, -2.552257, -0.759185, 1.570796, 1.904225],accel_mss,speed_ms,0,blend_radius_m)
    movel([0.329170, -1.402980, -2.550757, -0.758653, 1.570796, 1.899966],accel_mss,speed_ms,0,blend_radius_m)
    movel([0.328877, -1.403130, -2.550646, -0.758614, 1.570796, 1.899674],accel_mss,speed_ms,0,blend_radius_m)
    movel([0.328049, -1.403282, -2.550533, -0.758574, 1.570796, 1.898845],accel_mss,speed_ms,0,blend_radius_m)
    movel([0.327652, -1.403042, -2.550711, -0.758637, 1.570796, 1.898449],accel_mss,speed_ms,0,blend_radius_m)
    movel([0.327547, -1.402476, -2.551129, -0.758784, 1.570796, 1.898343],accel_mss,speed_ms,0,blend_radius_m)
    movel([0.327906, -1.401833, -2.551604, -0.758952, 1.570796, 1.898703],accel_mss,speed_ms,0,blend_radius_m)
    movel([0.328119, -1.401605, -2.551772, -0.759012, 1.570796, 1.898915],accel_mss,speed_ms,0,blend_radius_m)
    movel([0.331268, -1.398040, -2.554393, -0.759957, 1.570796, 1.902064],accel_mss,speed_ms,0,blend_radius_m)
    movel([0.332602, -1.396149, -2.555775, -0.760465, 1.570796, 1.903399],accel_mss,speed_ms,0,blend_radius_m)
    movel([0.333555, -1.394228, -2.557174, -0.760987, 1.570796, 1.904351],accel_mss,speed_ms,0,blend_radius_m)
    movel([0.333997, -1.392340, -2.558544, -0.761505, 1.570796, 1.904793],accel_mss,speed_ms,0,blend_radius_m)
    movel([0.334013, -1.390526, -2.559855, -0.762008, 1.570796, 1.904809],accel_mss,speed_ms,0,blend_radius_m)
    movel([0.333366, -1.387167, -2.562271, -0.762952, 1.570796, 1.904162],accel_mss,speed_ms,0,blend_radius_m)
    movel([0.333308, -1.386942, -2.562432, -0.763015, 1.570796, 1.904104],accel_mss,speed_ms,0,blend_radius_m)
    movel([0.333413, -1.386299, -2.562892, -0.763198, 1.570796, 1.904210],accel_mss,speed_ms,0,blend_radius_m)
    movel([0.333953, -1.385675, -2.563338, -0.763376, 1.570796, 1.904750],accel_mss,speed_ms,0,blend_radius_m)
    movel([0.334697, -1.385323, -2.563590, -0.763477, 1.570796, 1.905493],accel_mss,speed_ms,0,blend_radius_m)
    movel([0.335332, -1.385402, -2.563533, -0.763454, 1.570796, 1.906128],accel_mss,speed_ms,0,blend_radius_m)
    movel([0.335519, -1.385516, -2.563452, -0.763421, 1.570796, 1.906316],accel_mss,speed_ms,0,blend_radius_m)
    movel([0.338509, -1.387117, -2.562306, -0.762966, 1.570796, 1.909305],accel_mss,speed_ms,0,blend_radius_m)
    movel([0.340230, -1.387631, -2.561938, -0.762820, 1.570796, 1.911027],accel_mss,speed_ms,0,blend_radius_m)
    movel([0.342150, -1.387753, -2.561850, -0.762786, 1.570796, 1.912947],accel_mss,speed_ms,0,blend_radius_m)
    movel([0.344250, -1.387387, -2.562113, -0.762889, 1.570796, 1.915046],accel_mss,speed_ms,0,blend_radius_m)
    movel([0.346442, -1.386632, -2.562653, -0.763103, 1.570796, 1.917238],accel_mss,speed_ms,0,blend_radius_m)
    movel([0.350797, -1.384579, -2.564121, -0.763690, 1.570796, 1.921593],accel_mss,speed_ms,0,blend_radius_m)
    movel([0.351094, -1.384430, -2.564227, -0.763732, 1.570796, 1.921890],accel_mss,speed_ms,0,blend_radius_m)
    movel([0.351820, -1.384266, -2.564344, -0.763780, 1.570796, 1.922616],accel_mss,speed_ms,0,blend_radius_m)
    movel([0.352329, -1.384540, -2.564148, -0.763701, 1.570796, 1.923125],accel_mss,speed_ms,0,blend_radius_m)
    movel([0.352418, -1.385127, -2.563729, -0.763532, 1.570796, 1.923214],accel_mss,speed_ms,0,blend_radius_m)
    speed_ms = 0.003
    movel([0.352418, -1.378674, -2.560731, -0.772984, 1.570796, 1.923214],accel_mss,speed_ms,0,blend_radius_m)
    speed_ms = 0.05
    movel([0.352418, -1.353819, -2.548453, -0.810117, 1.570796, 1.923214],accel_mss,speed_ms,0,blend_radius_m)
    #M_RunCode9
    movel([0.376012, -1.090625, -2.686123, -0.935641, 1.570796, 1.946808],accel_mss,speed_ms,0,blend_radius_m)
    movel([0.376012, -1.031590, -2.645088, -1.035711, 1.570796, 1.946808],accel_mss,speed_ms,0,blend_radius_m)
    #M_RunCode2
    # End of main program
  end

  Machining2()
  $ 4 "Script: FaiChun_9 Jan_11_2_t3.script"
  def Machining3():
    # Default parameters:
    global speed_ms = 0.05
    global speed_rads = 0.75
    global accel_mss = 3
    global accel_radss = 1.2
    global blend_radius_m = 0.0003

